TYPE HVAC_SAFT :
STRUCT
	MesData				: HVAC ;	

	MesHygro_Amb		: REAL ; 		 (*(%)	 Hygro value*)
	MesTemp_Room		: REAL ; 		 (*(°C)	 Temperature value .*)
	MesTemp_Outside		: REAL ; 		 (*(°C)  Outside air temperature*)
	
	MesIDState			: WORD ; (* (NA) SubBankHVAC_St [SubBankHVAC_St] *) 

	
END_STRUCT
END_TYPE

(* stored: Version 1.1.0.1, ProductVersion 3.1.4024.6
   DUT HVAC_SAFT: Id {ff0351e3-f87b-4533-ac7c-6272149cace8} *)
